(* Logix 5000 project; controller Transcat_L33ER vendor 1 type 14 code 107 rev 32.11; software revision 32.02; part 4 of 4 *)
(* tags used below, declared in another part *)
   alwaysOFF : BOOL;
   AnyAutoDeviceInterlock : BOOL;   // Any device in Auto interlocked
   AnyAutoRun : BOOL;   // Bit that in on if ANY device is placed into Auto run (to signal pre-start beed)
   AnyDeviceInterlock : BOOL;   // Any device is interlocked
   AnyManualRun : BOOL;   // Bit that in on if ANY device is placed into manual run (to signal pre-start beed)
   Auto_Run_All_Interlock : BOOL;   // Bit to interlock all devices running in Auto
   BeaconBlueLight : ALIAS FOR TC_Remote_IO:3:O.3;   // Blue Beacon Light
   BeaconGreenLight : ALIAS FOR TC_Remote_IO:3:O.2;   // Green Beacon Light
   BeaconRedLight : ALIAS FOR TC_Remote_IO:3:O.0;   // Red Beacon Light
   BeaconYellowLight : ALIAS FOR TC_Remote_IO:3:O.1;   // Yellow Beacon Light
   Beep : BOOL;   // Bit to Activte Beacon Alarm
   BeepNew : ALIAS FOR TC_Remote_IO:3:O.4;
   Device : Device[20];
   FT103 : BronkhorstFlowMeter;
   FT103B : BronkhorstFlowMeter;
   FT104 : BronkhorstFlowMeter;
   FT104B : BronkhorstFlowMeter;
   FT105 : BronkhorstFlowMeter;
   FT105B : BronkhorstFlowMeter;
   GF101 : Thayer_WB_Feeder;   // Thayer 1 Tags
   GF201 : Thayer_WB_Feeder;   // Thayer 2 Tags
   GF301 : Acrison_Feeder;   // GF103 - Small Feeder 1
   GreenFlashingOff : TIMER;
   GreenFlashingOn : TIMER;
   HMI_AllReset : BOOL;   // Bit to reset Auto/Man, AutoRun, RecipeRun, TimedRunEnable to 0 from HMI
   HMI_ProcessReset : BOOL;   // Bit to clear the process hold/inteerlock when all other device interlocks are cleared
   MSG_FROM_SLC500 : INT[10];
   MX101 : Howes_Mixer;
   MX201 : Howes_Mixer;
   PT103_PV_RAW : ALIAS FOR TC_Remote_IO:1:I.Ch0Data;   // Raw (unscaled) pressure reading from PT103 - PSI * 100 (range 0 - 108 PSI)
   PT104_PV_RAW : ALIAS FOR TC_Remote_IO:1:I.Ch1Data;   // Raw (unscaled) pressure reading from PT104 - PSI * 100 (range 0 - 108 PSI)
   PT105_PV_RAW : ALIAS FOR TC_Remote_IO:1:I.Ch2Data;   // Raw (unscaled) pressure reading from PT105 - PSI * 100 (range 0 - 108 PSI)
   StartBeepTimer : TIMER;   // Timer to sound the beep alarm before starting a device
   UpperHowesSpeed : INT;
   VF101 : Acrison_Feeder;   // Medium Feeder Tags
   VF201 : Acrison_Feeder;   // Small Feeder 2 Tags
   VFD_Panel_Safety_Hoist_1_Cart_OK : ALIAS FOR XS26_VFD_Cabinet_Safety_Controller:I1.Data[2].2;   // HOIST 1 Cart Sensor
   VFD_Panel_Safety_Hoist_2_Cart_OK : ALIAS FOR XS26_VFD_Cabinet_Safety_Controller:I1.Data[2].3;   // HOIST 2 Cart Sensor
   YellowFlashOff : TIMER;
   YellowFlashOn : TIMER;
(* MainProgram, continued *)

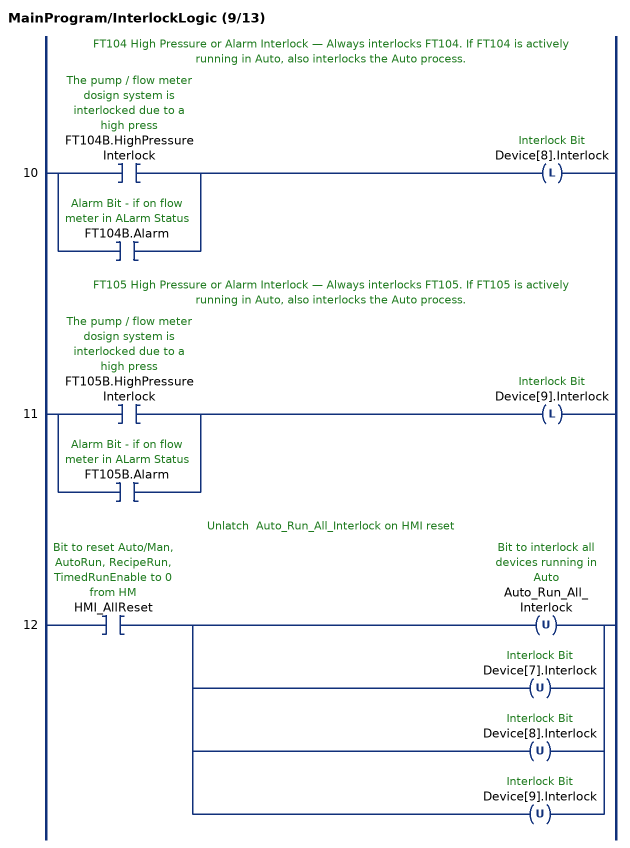
   // FT104 High Pressure or Alarm Interlock — Always interlocks FT104. If FT104 is actively running in Auto, also interlocks the Auto process.
   10: [XIC(FT104B.HighPressureInterlock) ,XIC(FT104B.Alarm) ]OTL(Device[8].Interlock);
   // FT105 High Pressure or Alarm Interlock — Always interlocks FT105. If FT105 is actively running in Auto, also interlocks the Auto process.
   11: [XIC(FT105B.HighPressureInterlock) ,XIC(FT105B.Alarm) ]OTL(Device[9].Interlock);
   // Unlatch  Auto_Run_All_Interlock on HMI reset
   12: XIC(HMI_AllReset)[OTU(Auto_Run_All_Interlock) ,[OTU(Device[7].Interlock) ,[OTU(Device[8].Interlock) ,OTU(Device[9].Interlock) ] ] ];
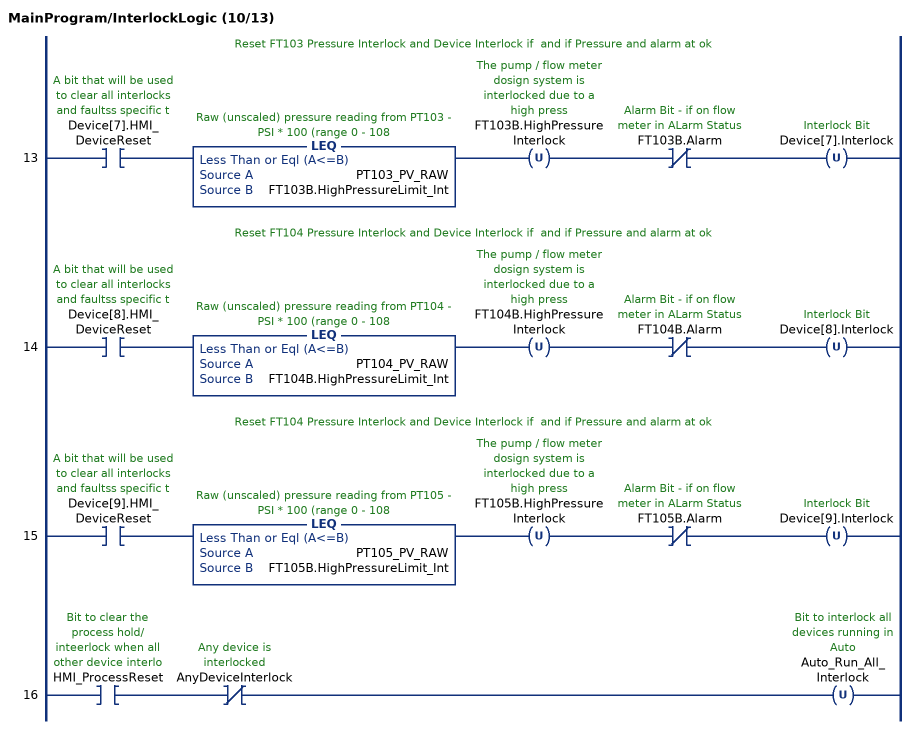
   // Reset FT103 Pressure Interlock and Device Interlock if  and if Pressure and alarm at ok
   13: XIC(Device[7].HMI_DeviceReset)LEQ(PT103_PV_RAW,FT103B.HighPressureLimit_Int)OTU(FT103B.HighPressureInterlock)XIO(FT103B.Alarm)OTU(Device[7].Interlock);
   // Reset FT104 Pressure Interlock and Device Interlock if  and if Pressure and alarm at ok
   14: XIC(Device[8].HMI_DeviceReset)LEQ(PT104_PV_RAW,FT104B.HighPressureLimit_Int)OTU(FT104B.HighPressureInterlock)XIO(FT104B.Alarm)OTU(Device[8].Interlock);
   // Reset FT104 Pressure Interlock and Device Interlock if  and if Pressure and alarm at ok
   15: XIC(Device[9].HMI_DeviceReset)LEQ(PT105_PV_RAW,FT105B.HighPressureLimit_Int)OTU(FT105B.HighPressureInterlock)XIO(FT105B.Alarm)OTU(Device[9].Interlock);
   16: XIC(HMI_ProcessReset)XIO(AnyDeviceInterlock)OTU(Auto_Run_All_Interlock);
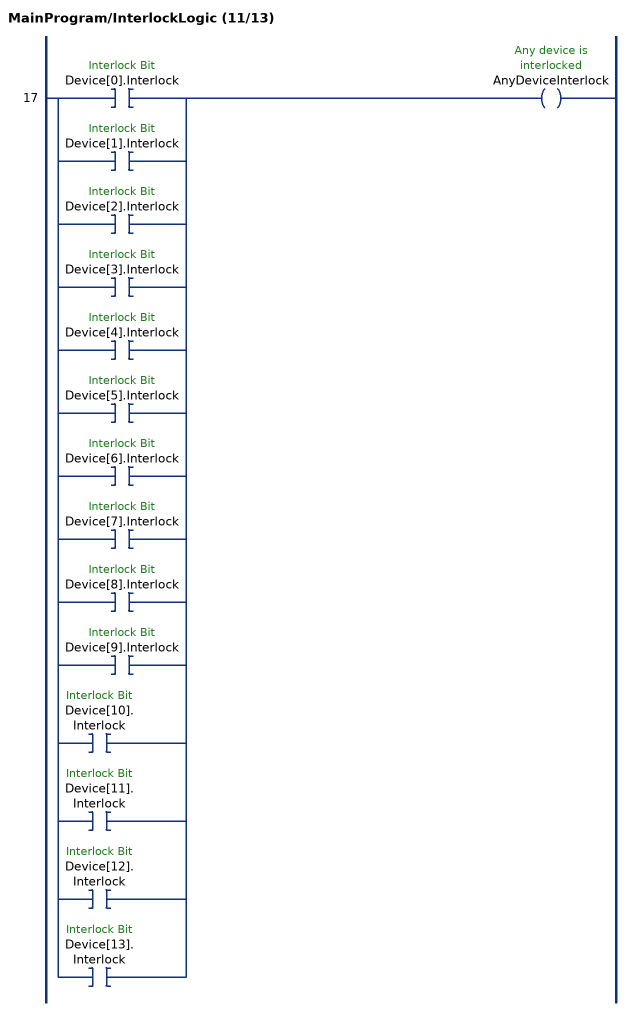
   17: [XIC(Device[0].Interlock) ,XIC(Device[1].Interlock) ,XIC(Device[2].Interlock) ,XIC(Device[3].Interlock) ,XIC(Device[4].Interlock) ,XIC(Device[5].Interlock) ,XIC(Device[6].Interlock) ,XIC(Device[7].Interlock) ,XIC(Device[8].Interlock) ,XIC(Device[9].Interlock) ,XIC(Device[10].Interlock) ,XIC(Device[11].Interlock) ,XIC(Device[12].Interlock) ,XIC(Device[13].Interlock) ]OTE(AnyDeviceInterlock);
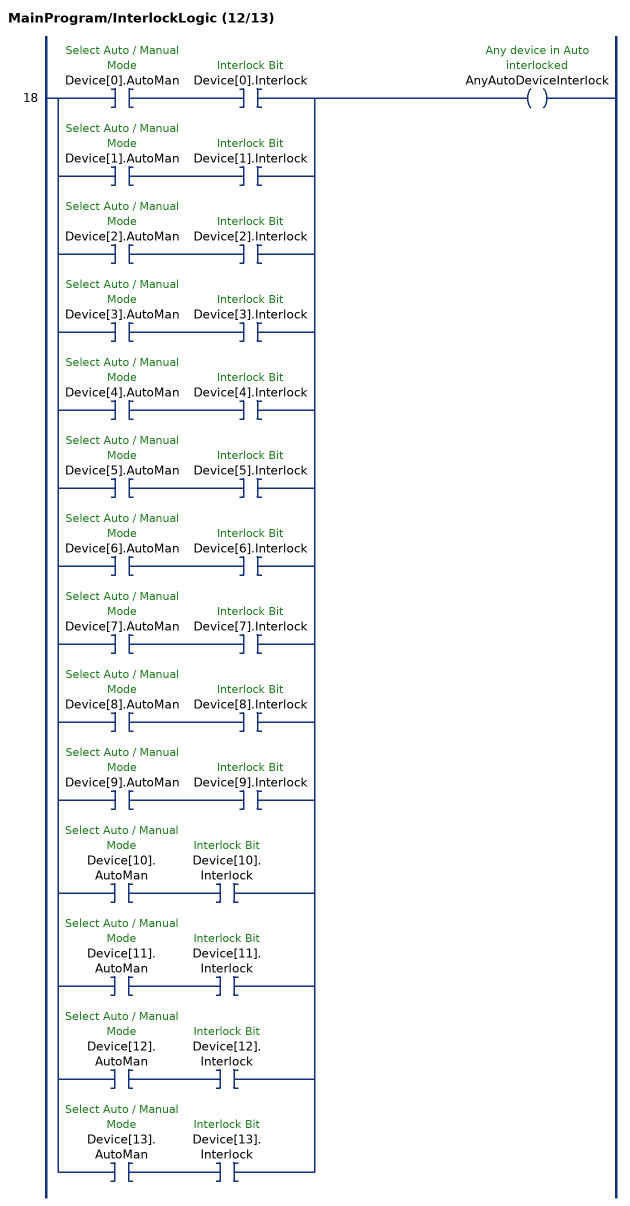
   18: [XIC(Device[0].AutoMan) XIC(Device[0].Interlock) ,XIC(Device[1].AutoMan) XIC(Device[1].Interlock) ,XIC(Device[2].AutoMan) XIC(Device[2].Interlock) ,XIC(Device[3].AutoMan) XIC(Device[3].Interlock) ,XIC(Device[4].AutoMan) XIC(Device[4].Interlock) ,XIC(Device[5].AutoMan) XIC(Device[5].Interlock) ,XIC(Device[6].AutoMan) XIC(Device[6].Interlock) ,XIC(Device[7].AutoMan) XIC(Device[7].Interlock) ,XIC(Device[8].AutoMan) XIC(Device[8].Interlock) ,XIC(Device[9].AutoMan) XIC(Device[9].Interlock) ,XIC(Device[10].AutoMan) XIC(Device[10].Interlock) ,XIC(Device[11].AutoMan) XIC(Device[11].Interlock) ,XIC(Device[12].AutoMan) XIC(Device[12].Interlock) ,XIC(Device[13].AutoMan) XIC(Device[13].Interlock) ]OTE(AnyAutoDeviceInterlock);
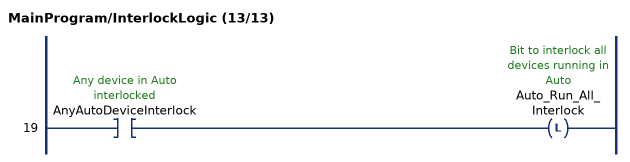
   19: XIC(AnyAutoDeviceInterlock)OTL(Auto_Run_All_Interlock);
END_ROUTINE

ROUTINE Light_Beacon   (* ladder *)
// Indicator Light Beacon
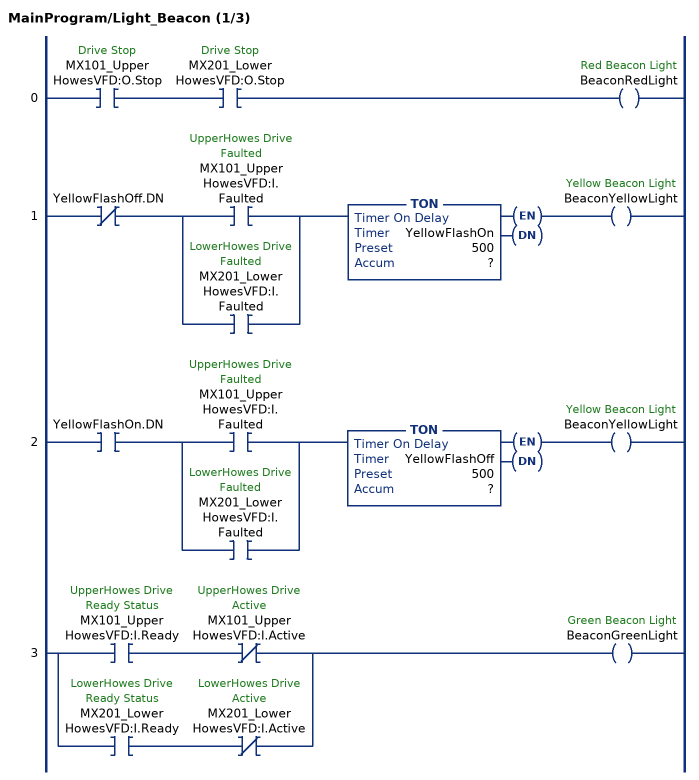
   0: XIC(MX101_UpperHowesVFD:O.Stop)XIC(MX201_LowerHowesVFD:O.Stop)OTE(BeaconRedLight);
   1: XIO(YellowFlashOff.DN)[XIC(MX101_UpperHowesVFD:I.Faulted) ,XIC(MX201_LowerHowesVFD:I.Faulted) ]TON(YellowFlashOn,?,?)OTE(BeaconYellowLight);
   2: XIC(YellowFlashOn.DN)[XIC(MX101_UpperHowesVFD:I.Faulted) ,XIC(MX201_LowerHowesVFD:I.Faulted) ]TON(YellowFlashOff,?,?)OTE(BeaconYellowLight);
   3: [XIC(MX101_UpperHowesVFD:I.Ready) XIO(MX101_UpperHowesVFD:I.Active) ,XIC(MX201_LowerHowesVFD:I.Ready) XIO(MX201_LowerHowesVFD:I.Active) ]OTE(BeaconGreenLight);
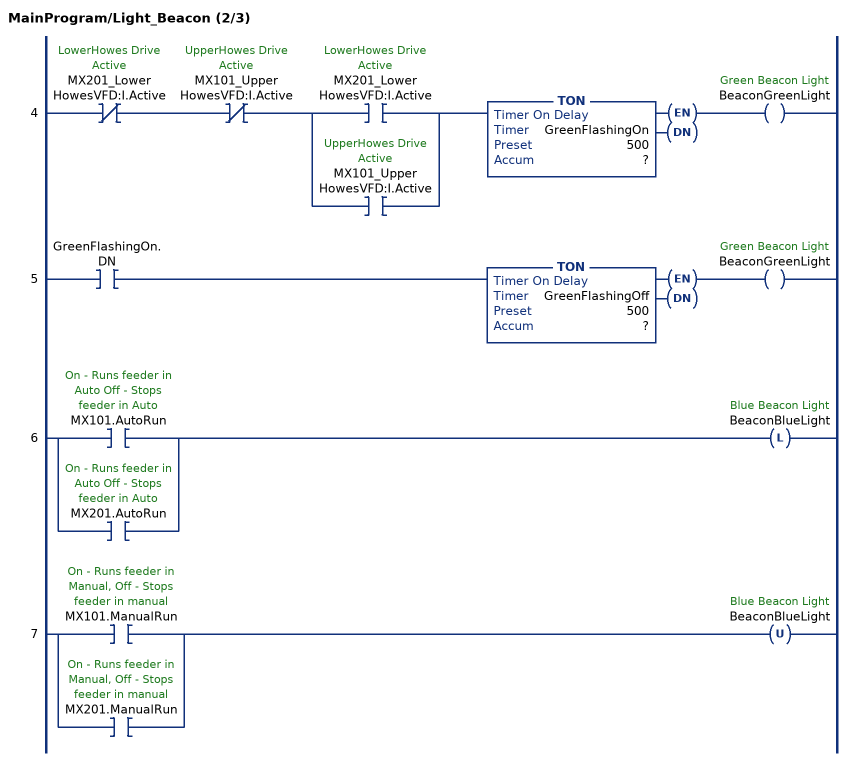
   4: XIO(MX201_LowerHowesVFD:I.Active)XIO(MX101_UpperHowesVFD:I.Active)[XIC(MX201_LowerHowesVFD:I.Active) ,XIC(MX101_UpperHowesVFD:I.Active) ]TON(GreenFlashingOn,?,?)OTE(BeaconGreenLight);
   5: XIC(GreenFlashingOn.DN)TON(GreenFlashingOff,?,?)OTE(BeaconGreenLight);
   6: [XIC(MX101.AutoRun) ,XIC(MX201.AutoRun) ]OTL(BeaconBlueLight);
   7: [XIC(MX101.ManualRun) ,XIC(MX201.ManualRun) ]OTU(BeaconBlueLight);
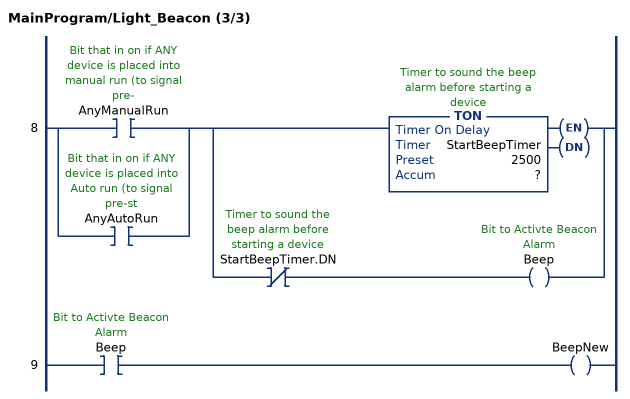
   8: [XIC(AnyManualRun) ,XIC(AnyAutoRun) ][TON(StartBeepTimer,?,?) ,XIO(StartBeepTimer.DN) OTE(Beep) ];
   9: XIC(Beep)OTE(BeepNew);
END_ROUTINE

ROUTINE MainRoutine   (* ladder *)
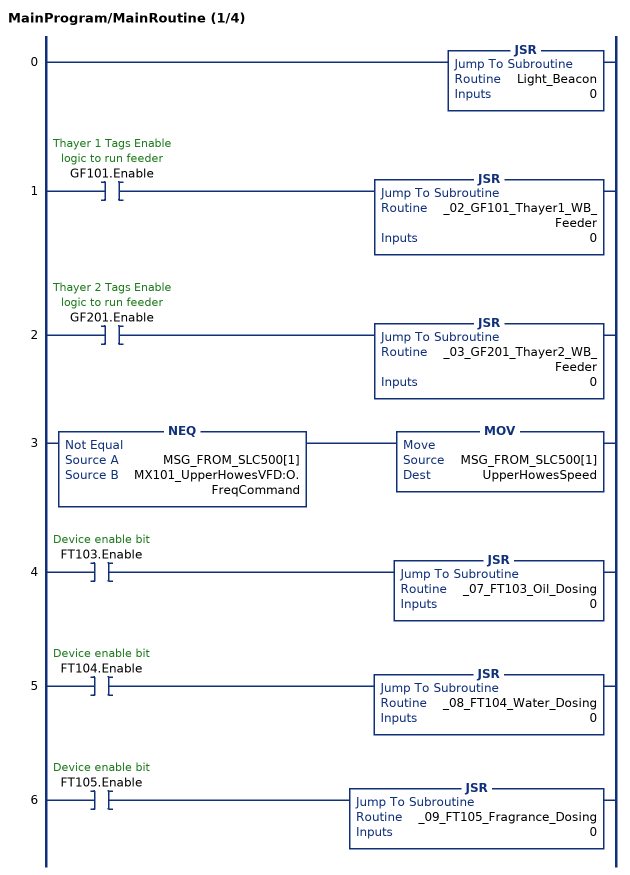
   0: JSR(Light_Beacon,0);
   1: XIC(GF101.Enable)JSR(_02_GF101_Thayer1_WB_Feeder,0);
   2: XIC(GF201.Enable)JSR(_03_GF201_Thayer2_WB_Feeder,0);
   3: NEQ(MSG_FROM_SLC500[1],MX101_UpperHowesVFD:O.FreqCommand)MOV(MSG_FROM_SLC500[1],UpperHowesSpeed);
   4: XIC(FT103.Enable)JSR(_07_FT103_Oil_Dosing,0);
   5: XIC(FT104.Enable)JSR(_08_FT104_Water_Dosing,0);
   6: XIC(FT105.Enable)JSR(_09_FT105_Fragrance_Dosing,0);
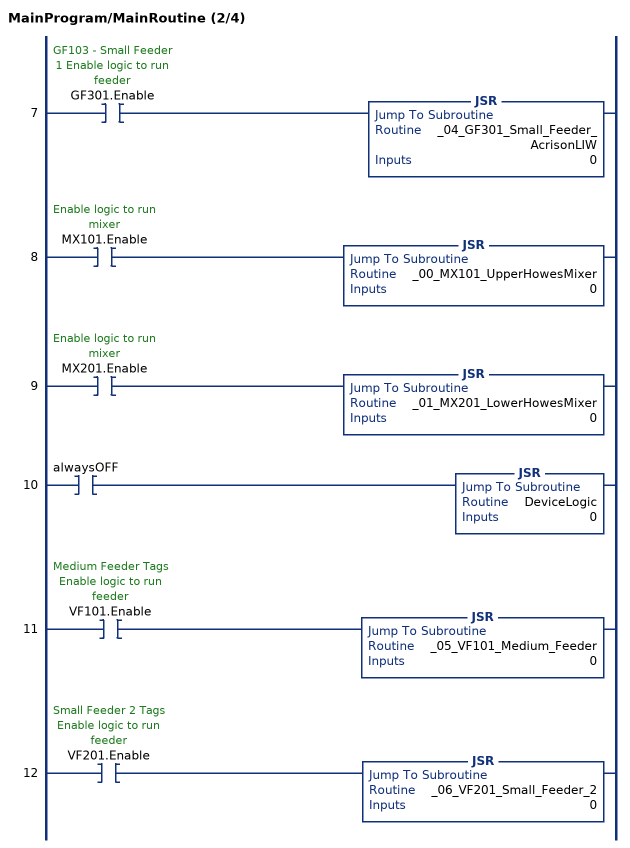
   7: XIC(GF301.Enable)JSR(_04_GF301_Small_Feeder_AcrisonLIW,0);
   8: XIC(MX101.Enable)JSR(_00_MX101_UpperHowesMixer,0);
   9: XIC(MX201.Enable)JSR(_01_MX201_LowerHowesMixer,0);
   10: XIC(alwaysOFF)JSR(DeviceLogic,0);
   11: XIC(VF101.Enable)JSR(_05_VF101_Medium_Feeder,0);
   12: XIC(VF201.Enable)JSR(_06_VF201_Small_Feeder_2,0);
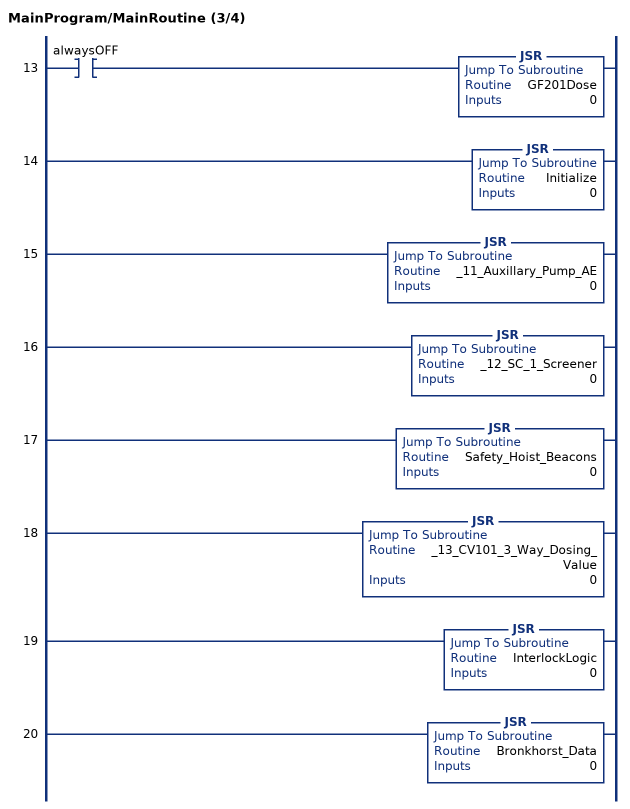
   13: XIC(alwaysOFF)JSR(GF201Dose,0);
   14: JSR(Initialize,0);
   15: JSR(_11_Auxillary_Pump_AE,0);
   16: JSR(_12_SC_1_Screener,0);
   17: JSR(Safety_Hoist_Beacons,0);
   18: JSR(_13_CV101_3_Way_Dosing_Value,0);
   19: JSR(InterlockLogic,0);
   20: JSR(Bronkhorst_Data,0);
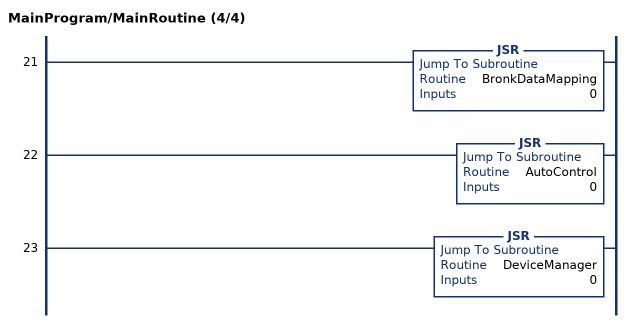
   21: JSR(BronkDataMapping,0);
   22: JSR(AutoControl,0);
   23: JSR(DeviceManager,0);
END_ROUTINE

ROUTINE Safety_Hoist_Beacons   (* ladder *)
// Saety Hoist Light Beacons
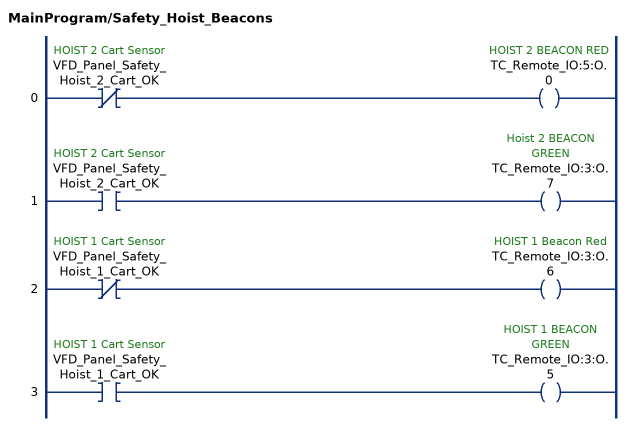
   0: XIO(VFD_Panel_Safety_Hoist_2_Cart_OK)OTE(TC_Remote_IO:5:O.0);
   1: XIC(VFD_Panel_Safety_Hoist_2_Cart_OK)OTE(TC_Remote_IO:3:O.7);
   2: XIO(VFD_Panel_Safety_Hoist_1_Cart_OK)OTE(TC_Remote_IO:3:O.6);
   3: XIC(VFD_Panel_Safety_Hoist_1_Cart_OK)OTE(TC_Remote_IO:3:O.5);
END_ROUTINE
END_PROGRAM
